// TIA Portal project "DawidKania_OptimizeReal" (V14)

(* hardware
DEVICE "S7-1200 station_1"  S7-1200 Station
   slot 0: "Rack_0"  S7-1200 Rack  Rack  V1.0
   slot 1: "PLC_1"  CPU 1214C DC/DC/DC  6ES7 214-1AG31-0XB0  V3.0
*)

// ===== PLC "PLC_1"  CPU 1214C DC/DC/DC =====

FUNCTION "OptimizedFunction" : Real   // FC1, SCL
{ S7_Optimized_Access := 'TRUE' }
VERSION : 0.1
   VAR_INPUT
      x1 : Real;
      x2 : Real;
   END_VAR
BEGIN
   // find minimum of function
   // y = x1 ^2 - 6 *x1 ^2.*x2 - 20 *x1 + 3 *x2 ^2 + 3 *x1 ^4 + 109


   #OptimizedFunction := #x1 ** REAL#2.0 - REAL#6.0 * #x1 ** REAL#2.0 * #x2 - REAL#20.0 * #x1 + REAL#3.0 * #x2 ** REAL#2.0 + REAL#3.0 * #x1 ** REAL#4.0 + REAL#109.0;
END_FUNCTION

FUNCTION "GradientSearchMin" : Real   // FC2, SCL
{ S7_Optimized_Access := 'TRUE' }
VERSION : 0.1
   VAR_INPUT
      x01 : Real;
      x02 : Real;
      iter : Int;
   END_VAR
   VAR_TEMP
      x1 : Real;
      x2 : Real;
      delta : Real;
      alpha : Real;
      y : Real;
      y1 : Real;
      y2 : Real;
      dy_dx1 : Real;
      dy_dx2 : Real;
   END_VAR
BEGIN

   #delta := REAL#0.001;
   #alpha := REAL#1.0;

   #x1 := #x01;
   #x2 := #x02;

   WHILE #iter >= 0 DO
       #iter := #iter - 1;

       // calculate gradient
       #y := "OptimizedFunction"(x1:=#x1, x2:=#x2);
       #y1 := "OptimizedFunction"(x1:=#x1 + #delta, x2:=#x2);
       #y2 := "OptimizedFunction"(x1:=#x1, x2:=#x2 + #delta);

       #dy_dx1 := (#y1 - #y) / #delta;
       #dy_dx2 := (#y2 - #y) / #delta;

       #x1 := #x1 - #alpha * #dy_dx1;
       #x2 := #x2 - #alpha * #dy_dx2;

   END_WHILE;

   #GradientSearchMin := "OptimizedFunction"(x1:=#x1, x2:=#x2);
END_FUNCTION

ORGANIZATION_BLOCK "Main"   // OB1, SCL, ProgramCycle
TITLE = "Main Program Sweep (Cycle)"
{ S7_Optimized_Access := 'TRUE' }
VERSION : 0.1
   VAR_TEMP
      minimum : Real;
   END_VAR
BEGIN


   #minimum := "GradientSearchMin"(x01:=REAL#100.0, x02:=REAL#100.0, iter:=1000);
END_ORGANIZATION_BLOCK